TYPE (* Telemetry connection health: wraps the MQTT_CONNECTION status outputs *)
  (* Standard: 1131-3 *)
  (* Version 0.1, 6/21/2026, easensoy, WMG, single STRUCT output for Telemetry *)
  PACKAGE Main;
  TelemetryHealth : STRUCT
    IsConnected : BOOL;
    ReturnCode : USINT;
    Status : STRING[255];
    NetworkState : STRING[80];
    SecurityState : STRING[80];
    ProtocolState : STRING[80];
  END_STRUCT;
END_TYPE
